% RSLogix 500 project I2P HANDOUT 05_BAK024.RSS, saved by version 10.00.00.00 %
PROJECT "UNTITLED"    % processor: Bul.1763 MicroLogix 1100 Series B %

PROGRAM FILES
  LAD 2   6 rungs

DATA FILES
  O0 OUTPUT  4 elements
  I1 INPUT  6 elements
  S2 STATUS  66 elements
  B3 BINARY  2 elements
  T4 TIMER  2 elements
  C5 COUNTER  1 elements
  R6 CONTROL  1 elements
  N7 INTEGER  1 elements
  F8 FLOAT  2 elements

LADDER 2
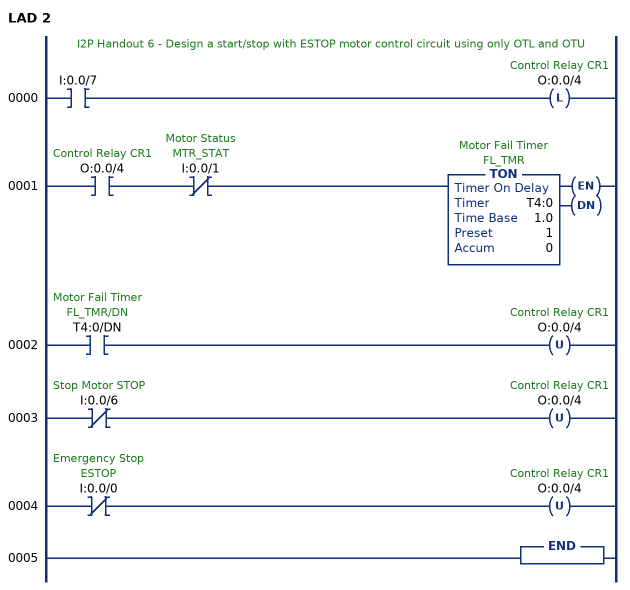
% Rung: 0 %
% I2P Handout 6 - Design a start/stop with ESTOP motor control circuit using only OTL and OTU %
SOR XIC I:0.0/7 OTL O:0.0/4 EOR
%   O:0.0/4  CR1  "Control Relay" %
% Rung: 1 %
SOR XIC O:0.0/4 XIO I:0.0/1 TON T4:0 1.0 1 0 EOR
%   O:0.0/4  CR1  "Control Relay" %
%   I:0.0/1  MTR_STAT  "Motor Status" %
%   T4:0  FL_TMR  "Motor Fail Timer" %
% Rung: 2 %
SOR XIC T4:0/DN OTU O:0.0/4 EOR
%   T4:0  FL_TMR  "Motor Fail Timer" %
%   O:0.0/4  CR1  "Control Relay" %
% Rung: 3 %
SOR XIO I:0.0/6 OTU O:0.0/4 EOR
%   I:0.0/6  STOP  "Stop Motor" %
%   O:0.0/4  CR1  "Control Relay" %
% Rung: 4 %
SOR XIO I:0.0/0 OTU O:0.0/4 EOR
%   I:0.0/0  ESTOP  "Emergency Stop" %
%   O:0.0/4  CR1  "Control Relay" %
% Rung: 5 %
SOR END EOR

OTHER DOCUMENTED ADDRESSES
  B3:0/0  MTR_CMD  "Motor Command"
  FALSE  

DATA TABLE (non-zero values as saved)
DATA B3
% B3:0 % 0X0002 0X0000
DATA T4
% .PRE .ACC %
% T4:0 % 1 0
DATA C5
% .PRE .ACC %
% C5:0 % 5 0
DATA N7
% N7:0 % 10
